(* Schneider Machine Expert - Basic project PID, file version 2.7.0.0 *)
(* ProjectInformations: Name=Nuevo proyecto *)

HARDWARE
  Cpu 0: TM221M16R/G
  EthernetConfiguration: NetworkName=M221, IpAllocationMode=FixedAddress, IpAddress=0.0.0.0, SubnetMask=0.0.0.0
  SerialLineConfiguration: Baud=Baud19200, Parity=ParityEven, DataBits=DataBits8, StopBits=StopBits1, PhysicalMedium=PhysicalMediumRs485, TransmissionMode=TransmissionModeModbusRtu, SlaveId=1, Addressing=SlaveAddressing
  MastTask: UsePeriodScanMode=true, PeriodScan=50
  FastTask: Period=255
  CpuBehavior: StartingMode=StartAsPreviousState, AutoSaveRamOnEeprom=true, WatchdogPeriod=250

SYMBOLS  (address, symbol, comment, settings)
  %M0       AT_TRIGGER
  %M7       TRIGGER
  %M8       INVERSE
  %M500     PID_ACTIVE
  %MW1      FLOW_MESURE
  %MW2      SET_POINT
  %MW3      FILL_VALVE
  %MW5      SET_POINT_VIEW
  %MW6      FLOW_VIEW
  %MW100    STATES
  %MW200    KP
  %MW300    TI
  %MW400    TD

POU Nuevo POU
  (* SectionNumber=1 *)

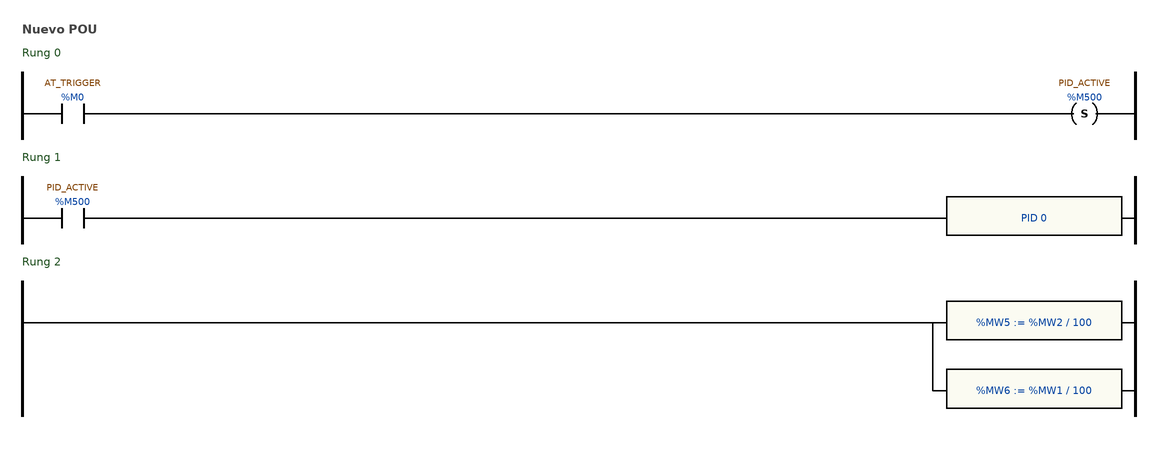

// Rung 0
  LD %M0                  (* AT_TRIGGER *)
  S %M500                 (* PID_ACTIVE *)
  // as ST:
  //   IF AT_TRIGGER THEN PID_ACTIVE := TRUE; END_IF;

// Rung 1
  LD %M500                (* PID_ACTIVE *)
  [ PID 0 ]
  // as ST:
  //   IF PID_ACTIVE THEN PID 0; END_IF;

// Rung 2
  LD 1
  [ %MW5 := %MW2 / 100 ]  (* SET_POINT_VIEW, SET_POINT *)
  [ %MW6 := %MW1 / 100 ]  (* FLOW_VIEW, FLOW_MESURE *)
  // as ST:
  //   SET_POINT_VIEW := SET_POINT / 100;
  //   FLOW_VIEW := FLOW_MESURE / 100;
